(* Schneider Machine Expert - Basic project Y=A'(B+CD), file version 2.9.0.0 *)
(* ProjectInformations: Name=New project *)

HARDWARE
  Cpu 0: TM221CE24R
  EthernetConfiguration: NetworkName=M221, IpAllocationMode=FixedAddress, IpAddress=0.0.0.0, SubnetMask=0.0.0.0
  SerialLineConfiguration: Baud=Baud19200, Parity=ParityEven, DataBits=DataBits8, StopBits=StopBits1, PhysicalMedium=PhysicalMediumRs485, SlaveId=1, Addressing=SlaveAddressing
  MastTask: UsePeriodScanMode=false, PeriodScan=100
  FastTask: Period=255
  CpuBehavior: StartingMode=StartAsPreviousState, AutoSaveRamOnEeprom=true, WatchdogPeriod=250

SYMBOLS  (address, symbol, comment, settings)
  %I0.0     A
  %I0.1     B
  %I0.2     C
  %I0.3     DS
  %Q0.0     Y

POU New POU
  (* SectionNumber=1 *)

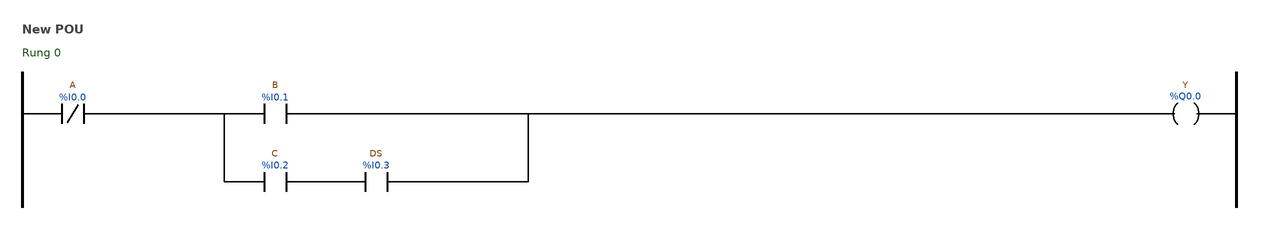

// Rung 0
  LDN %I0.0               (* A *)
  AND( %I0.1              (* B *)
  OR( %I0.2               (* C *)
  AND %I0.3               (* DS *)
  )
  )
  ST %Q0.0                (* Y *)
  // as ST:
  //   Y := NOT A AND (B OR C AND DS);
